PROGRAM MAIN
VAR
END_VAR

END_PROGRAM

(* stored: Version 1.1.0.1
   POU MAIN: Id {61be8268-078e-44ff-8840-b308aec80eef} *)
